PROGRAM SafetyHandling
VAR
	state           : INT := 0;            
	// power on delay
	start_delay 	: TON := (PT := T#2S);
	state_delay 	: TON := (PT := T#1S);

	// Safety group
	fbInfoGroup1			:FB_InfoGroup;
	stInfoGroup1	AT%I*	:ST_InfoDataGroup;
	sStateGroup1			:STRING;
	
	// Estop
	fbInfoEStop1			:FB_InfoEStop;
	stInfoEStop1 	AT%I*	:ST_InfoDataFB;
	sStateEStop1			:STRING;
	sDiagEStop1				:STRING;	
	
	// Info EL1904
	fbInfoSafetyIn			:FB_InfoConnection;
	stInfoSafetyIn 	AT%I*	:ST_InfoDataConnection;
	sStateSafetyIn			:STRING;
	sDiagSafetyIn			:STRING;
	bSafetyInCh1			:BOOL;
	bSafetyInCh2			:BOOL;
	bSafetyInCh3			:BOOL;
	bSafetyInCh4			:BOOL;
	
	// Info EL2904
	fbInfoSafetyOut			:FB_InfoConnection;
	stInfoSafetyOut AT%I*	:ST_InfoDataConnection;
	sStateSafetyOut			:STRING;
	sDiagSafetyOut			:STRING;
	bSafetyOutCh1			:BOOL;
	bSafetyOutCh2			:BOOL;
	bSafetyOutCh3			:BOOL;
	bSafetyOutCh4			:BOOL;
	
	// Errack logging
	ErrAckLog		: FB_EventLog;
	// restart logging
	RestartLog		: FB_EventLog;
	// safety logging
	SafetyLog		: FB_EventLog;
	
END_VAR
VAR_OUTPUT
	// error condition
	Error			: BOOL;
	// Emergency_stop engaged
	Emergency_stop	: BOOL;
END_VAR
VAR_INPUT
	// issue a remote restart
	remote_restart:		BOOL;
	// issue a remute run/stop
	remote_run:			BOOL := TRUE;
END_VAR

// Safety is running on start
GVL_Safety.Run := remote_run;

fbInfoGroup1(
	stInfoData	:= stInfoGroup1,
	sState		=> sStateGroup1);

fbInfoEStop1(
	stInfoData	:= stInfoEStop1, 
	sState		=> sStateEStop1, 
	sDiag		=> sDiagEStop1);

//Info SafetyIn EL1904
fbInfoSafetyIn(
	stInfoData		:=stInfoSafetyIn, 
	sState			=>sStateSafetyIn, 
	sDiag			=>sDiagSafetyIn, 
	bChannel1		=>bSafetyInCh1, 
	bChannel2		=>bSafetyInCh2, 
	bChannel3		=>bSafetyInCh3, 
	bChannel4		=>bSafetyInCh4);	
	
//Info SafetyOut EL2904
fbInfoSafetyOut(
	stInfoData		:=stInfoSafetyOut, 
	sState			=>sStateSafetyOut, 
	sDiag			=>sDiagSafetyOut, 
	bChannel1		=>bSafetyOutCh1, 
	bChannel2		=>bSafetyOutCh2, 
	bChannel3		=>bSafetyOutCh3, 
	bChannel4		=>bSafetyOutCh4);
	
(*

// power on delay for Safety RESTART after RUN=1
start_delay(IN := TRUE);

CASE state OF
	0:
	    IF start_delay.Q  THEN
			GVL_Safety.ErrAck := TRUE;
			state := 1;
		END_IF
	1:
		state_delay(IN := TRUE);	
		IF state_delay.Q THEN
			GVL_Safety.ErrAck := FALSE;
			GVL_Safety.Restart := TRUE;
			state := 2;
			state_delay(IN := FALSE);
		END_IF
	2:
		state_delay(IN := TRUE);	
		IF state_delay.Q THEN
			GVL_Safety.Restart := FALSE;
			GVL_Safety.ErrAck := TRUE;
			state := 3;
			state_delay(IN := FALSE);
		END_IF
	3:
		state_delay(IN := TRUE);	
		IF state_delay.Q THEN	
			GVL_Safety.ErrAck := FALSE;
			state := 4;
			state_delay(IN := FALSE);
		END_IF	
END_CASE

// remote restart
IF remote_restart THEN
	state := 0;
	remote_restart := FALSE;
END_IF

// manual Err_Ack 
GVL_Safety.ErrAck := (GVL_Main.key_switch_remote AND GVL_Main.reset_switch);

// manual Restart
GVL_Safety.Restart := (GVL_Main.key_switch_remote AND GVL_Main.start_switch);

ErrAckLog(	Trigger := GVL_Safety.ErrAck,
			OnMessage := 'Safety error was acknowledged.');
			
RestartLog(	Trigger := GVL_Safety.Restart,
			Level := ADSLOG_MSGTYPE_WARN,
			OnMessage := 'Safety was restarted.');

SafetyLog(	Trigger := Error,
			Level := ADSLOG_MSGTYPE_ERROR,
			OnMessage := 'Safety Error! Emergency stop enganged!',
			OffMessage := 'Safety is OK.',
			OffLevel := ADSLOG_MSGTYPE_HINT);
*)

(*
// wait n seconds after Start ...
start_delay(IN := TRUE);
// ... and send ErrAck for n milliseconds
ErrAck_Pulse(IN := (GVL_Safety.State = 2) AND start_delay.Q);

// Error Acknowledgment: Turn key_switch OFF and press STOP 
GVL_Safety.ErrAck := (GVL_Main.key_switch_remote AND GVL_Main.reset_switch)
					OR ErrAck_Pulse.Q
					OR remote_ErrAck;
// detect falling edge 
ErrAck_Trigger(CLK := GVL_Safety.ErrAck);
// send restart pulse on falling edge of ErrAck
restart_pulse(IN := ErrAck_Trigger.Q);

// RESTART Safety after pushing reset or power on delay
GVL_Safety.Restart := (GVL_Main.key_switch_remote AND GVL_Main.start_switch)
 					   OR remote_restart
                       OR restart_pulse.Q;
				
//Error := GVL_Safety.Error OR (GVL_Safety.State <> 1);

//Emergency_stop := NOT GVL_Safety.Stop;

ErrAckLog(	Trigger := GVL_Safety.ErrAck,
			OnMessage := 'Safety error was acknowledged.');
			
RestartLog(	Trigger := GVL_Safety.Restart,
			Level := ADSLOG_MSGTYPE_WARN,
			OnMessage := 'Safety was restarted.');

SafetyLog(	Trigger := Error,
			Level := ADSLOG_MSGTYPE_ERROR,
			OnMessage := 'Safety Error! Emergency stop enganged!',
			OffMessage := 'Safety is OK.',
			OffLevel := ADSLOG_MSGTYPE_HINT);
*)

END_PROGRAM

(* stored: Version 1.1.0.1, ProductVersion 3.1.4024.12
   POU SafetyHandling: Id {6d4a788c-2168-4769-93de-c67314036861}, SpecialFunc None *)
